FUNCTION_BLOCK Forces4
VAR_INPUT
END_VAR
VAR_OUTPUT
END_VAR
VAR
END_VAR

END_FUNCTION_BLOCK

(* stored: Version 1.1.0.1, ProductVersion 3.1.4024.11
   POU Forces4: Id {d56f4d88-04e3-4b2c-89b6-4800afcabbe7}, SpecialFunc None *)
